TYPE E_CameraRegisters :
(
pDeviceManifestSchemaMinorVersionReg_pDeviceManifestXMLMajorVersionReg_DeviceManifestSecondaryURL_pDeviceManifestSchemaMajorVersionReg_pDeviceManifestXMLSubMinorVersionReg_pDeviceManifestXMLMinorVersionReg_DeviceManifestPrimaryURL_BootStrap_VersionMajor_BootStrap_VersionMinor := 16#00000000, // GigE Vision Minor Version
BootStrap_DeviceEndianess_BootStrap_CharacterSet_pURLRegisterAddressReg := 16#00000004, // None
BootStrap_MACAddress_High      := 16#00000008, // None
BootStrap_MACAddress_Low       := 16#0000000C, // None
BootStrap_EnabledDHCP_BootStrap_EnabledPersistentIP_BootStrap_EnabledLLA := 16#00000014, // LLA Register Enabled
BootStrap_IPAddress            := 16#00000024, // Current IP Address Register
BootStrap_SubnetMask           := 16#00000034, // Current Subnet Mask Register
BootStrap_Gateway              := 16#00000044, // Current Subnet Mask Register
DeviceVendorName               := 16#00000048, // Name of the camera vendor which is always Beckhoff Automation GmbH & Co.KG
DeviceModelName                := 16#00000068, // Displays the device model name.
DeviceVersion                  := 16#00000088, // Displays the device version which includes the firmware release and build.
DeviceSerialNumber             := 16#000000D8, // Device's serial number. This string is a unique identifier of the device.
DeviceUserID                   := 16#000000E8, // A user set ID of up to 15 characters. By default this field is set to the serial number of the camera.
GevFirstURL                    := 16#00000200, // NULL-terminated string providing the first URL to the XML device description file.
GevSecondURL                   := 16#00000400, // NULL-terminated string providing the second URL to the XML device description file.
BootStrap_NumberOfInterfaces   := 16#00000600, // Number Of Interfaces
BootStrap_PersistentIPAddress  := 16#0000064C, // Persistent IP Address Register
BootStrap_PersistentSubnetMask := 16#0000065C, // Persistent Subnet Mask Register
BootStrap_PersistentDefaultGateway := 16#0000066C, // Persistent Default Gateway Register
BootStrap_TimestampTickFrequencyHigh := 16#0000093C, // 32-MSB of the timestamp Frequency
BootStrap_TimestampTickFrequencyLow := 16#00000940, // 32-LSB of the timestamp Frequencyy
BootStrap_GevTimestampControl  := 16#00000944, // Timestamp Control Register
BootStrap_TimestampValueHigh   := 16#00000948, // 32-MSB of the timestamp Value
BootStrap_TimestampValueLow    := 16#0000094C, // 32-LSB of the timestamp Value
pGevDiscoveryAckDelayReg       := 16#00000950, // Gev Discovery Ack Delay register
BootStrap_GVSPExtendedID       := 16#00000960, // GVSP Extended ID
BootStrap_StreamChannelDestinationPort := 16#00000D00, // BootStrap Stream Channel Destination Port register
pGevSCPSDoNotFragmentReg       := 16#00000D04, // None
pGevSCPDReg                    := 16#00000D08, // Inter-Packet Delay Register
BootStrap_StreamChannelDestinationAddress := 16#00000D18, // BootStrap Stream Channel Destination Address register
BootStrap_StreamChannelSourcePort := 16#00000D1C, // BootStrap Stream Channel Source Port register
pReverseXReg                   := 16#01F81400, // None
pAcquisitionModeReg            := 16#01F83200, // None
pGevPhysicalLinkConfiguration  := 16#01F84E00, // None
pDeviceTypeReg                 := 16#01F90000, // None
pAcquisitionFrameRateEnableIsAvailableReg := 16#01F93400, // None
pEtherCATLinkActiveReg         := 16#01F93900, // None
pPayloadSizeHighReg            := 16#01F93D00, // None
pPayloadSizeLowReg             := 16#01F93D04, // None
pGevActiveLinkCountReg         := 16#01F93E00, // None
pOpticControllerPresentReg     := 16#01F94500, // None
pLightControllerPresentReg     := 16#01F95200, // None
pTestPatternCountReg           := 16#01FA0204, // None
pOpticControllerStatusReg      := 16#01FA1100, // None
pLightControllerPowerGoodReg   := 16#01FA1300, // None
pReverseYReg                   := 16#02F81400, // None
pAcquisitionStartReg           := 16#02F83200, // None
pGainBaseReg                   := 16#02F84600, // None
pDigitalAllGainReg             := 16#02F84604, // None
pDigitalRedGainReg             := 16#02F84608, // None
pDigitalGreenGainReg           := 16#02F8460C, // None
pDigitalBlueGainReg            := 16#02F84610, // None
pGevCurrentPhysicalLinkConfiguration := 16#02F84E00, // None
pTemperatureCompensationModeReg := 16#02F86C00, // None
pLightControllerEnabledReg     := 16#02F87D00, // None
pDeviceScanTypeReg             := 16#02F90000, // None
pAcquisitionFrameRateIsAvailableReg := 16#02F93400, // None
pEtherCATStateReg              := 16#02F93900, // None
pTransferBlockDurationHighReg  := 16#02F93B00, // None
pTransferBlockDurationLowReg   := 16#02F93B04, // None
pApertureReg                   := 16#02F94500, // Aperture Register
pLightConnectionStatusReg      := 16#02F95200, // None
pDeviceTemperatureImageSensorReg := 16#02FA0000, // None
pDeviceTemperatureCoreReg      := 16#02FA0004, // None
pDeviceTemperatureEthernetPhyReg := 16#02FA0008, // None
pDeviceTemperatureLiquidLensReg := 16#02FA000C, // None
TestPatternDescription         := 16#02FA0200, // None
pLightController0Channel0TriggerActiveReg := 16#02FA1300, // Trigger selected channel active register
pLightController0Channel1TriggerActiveReg := 16#02FA1304, // Trigger channel 1 active register
pLightController0Channel2TriggerActiveReg := 16#02FA1308, // Trigger channel 2 active register
pLightController0Channel3TriggerActiveReg := 16#02FA130C, // Trigger channel 3 active register
pPixelFormatReg                := 16#03F81400, // None
pAcquisitionStopReg            := 16#03F83200, // None
pMinimumObjectCameraDistanceReg := 16#03F83504, // Minimum Object Camera Distance Register
pMaximumObjectCameraDistanceReg := 16#03F83508, // Maximum Object Camera Distance Register
pObjectCameraDistanceReg       := 16#03F86C00, // Object Camera Distance Register
pPhysicalWidthReg              := 16#03F92600, // None
pGevSupportedOptionHighWordReg := 16#03F93E00, // None
pGevSupportedOptionLowWordReg  := 16#03F93E04, // None
pNumericalApertureReg          := 16#03F94500, // Numerical Aperture Register
pTestPatternReg                := 16#03FA0200, // None
pDecimationImplementedReg      := 16#04F81400, // None
pDecimationModesCapabilityReg  := 16#04F81404, // None
pDecimationHorizontalFactorsCapabilityReg := 16#04F81408, // None
pDecimationVerticalFactorsCapabilityReg := 16#04F8140C, // None
pAcquisitionAbortReg           := 16#04F83200, // None
pBlackLevelReg                 := 16#04F84600, // None
pGevPAUSEFrameReception        := 16#04F84E00, // None
pLensCalibrationModeReg        := 16#04F86C00, // Lens Calibration Mode Register
LightController0Channel0ColorDescription := 16#04F87D00, // The color of the emitted light.
LightController0Channel1ColorDescription := 16#04F87D20, // The color of the emitted light.
LightController0Channel2ColorDescription := 16#04F87D40, // The color of the emitted light.
LightController0Channel3ColorDescription := 16#04F87D60, // The color of the emitted light.
pPhysicalHeightReg             := 16#04F92600, // None
pAcquisitionStatusAcquisitionTriggerWaitReg := 16#04F93400, // None
pAcquisitionStatusAcquisitionActiveReg := 16#04F93404, // None
pGevMACAddressHighWordReg      := 16#04F93E00, // None
pFocalPowerReg                 := 16#04F94500, // Focal Power Register
pTestPatternModeReg            := 16#04FA0200, // None
pDeviceLink0ThroughputLimitModeReg := 16#05F80000, // None
pDeviceLink1ThroughputLimitModeReg := 16#05F80040, // None
pDecimationHorizontalModeReg   := 16#05F81400, // None
pAcquisitionFrameCountReg      := 16#05F83200, // None
pBlackLevelAutoReg             := 16#05F84600, // None
pGevPAUSEFrameTransmission     := 16#05F84E00, // None
pLensCalibrationStepNearReg    := 16#05F86C00, // None
pLightController0Channel0BrightnessReg := 16#05F87D00, // Light Controller0 Channel0 Brightness register
pLightController0Channel1BrightnessReg := 16#05F87D04, // Light Controller0 Channel1 Brightness register
pLightController0Channel2BrightnessReg := 16#05F87D08, // Light Controller0 Channel2 Brightness register
pLightController0Channel3BrightnessReg := 16#05F87D0C, // Light Controller0 Channel3 Brightness register
DeviceFamilyName               := 16#05F90000, // Displays the family of the camera model.
pSensorPixelWidthReg           := 16#05F92600, // None
pLineTriggerAvailableReg       := 16#05F93400, // None
pGevMACAddressLowWordReg       := 16#05F93E00, // None
pObjectSensorDistanceReg       := 16#05F94500, // Object Sensor Distance Register
pTestPatternParameter1Reg      := 16#05FA0200, // None
pDeviceLink0ThroughputLimitRatioReg := 16#06F80000, // None
pDeviceLink1ThroughputLimitRatioReg := 16#06F80040, // None
pDeviceLinkMinimumThroughputLimitRatioReg := 16#06F80044, // None
pDecimationHorizontalReg       := 16#06F81400, // None
pAcquisitionFrameRateEnableReg := 16#06F83200, // None
pLensCalibrationStepFarReg     := 16#06F86C00, // None
pLightController0Channel0BrightnessMinimumReg := 16#06F87D00, // Light Controller0 Channel0 Brightness Minimum register
pLightController0Channel1BrightnessMinimumReg := 16#06F87D04, // Light Controller0 Channel1 Brightness Minimum register
pLightController0Channel2BrightnessMinimumReg := 16#06F87D08, // Light Controller0 Channel2 Brightness Minimum register
pLightController0Channel3BrightnessMinimumReg := 16#06F87D0C, // Light Controller0 Channel3 Brightness Minimum register
DeviceManufacturerInfo         := 16#06F90000, // Manufactuer information about the device.
pSensorPixelHeightReg          := 16#06F92600, // None
pGevIPConfigurationStatusReg   := 16#06F93E00, // None
pFocalLengthReg                := 16#06F94500, // Focal Length Register
pTestPatternParameter2Reg      := 16#06FA0200, // None
pDeviceLink0ThroughputLimitReg := 16#07F80000, // None
pDeviceLink1ThroughputLimitReg := 16#07F80040, // None
pDecimationHorizontalMinimumReg := 16#07F81400, // None
pFrameRateReg                  := 16#07F83200, // None
pBalanceRatioReg               := 16#07F84600, // None
pBalanceRatioRedReg            := 16#07F84604, // None
pBalanceRatioGreenReg          := 16#07F84608, // None
pBalanceRatioBlueReg           := 16#07F8460C, // None
pLensCalibrationCoefficient1Reg := 16#07F86C00, // Lens Calibration Coefficient 1 Register
pLightController0Channel0BrightnessMaximumReg := 16#07F87D00, // Light Controller0 Channel0 Brightness Maximum register
pLightController0Channel1BrightnessMaximumReg := 16#07F87D04, // Light Controller0 Channel1 Brightness Maximum register
pLightController0Channel2BrightnessMaximumReg := 16#07F87D08, // Light Controller0 Channel2 Brightness Maximum register
pLightController0Channel3BrightnessMaximumReg := 16#07F87D0C, // Light Controller0 Channel3 Brightness Maximum register
SensorName                     := 16#07F92600, // Displays the model of the sensor.
pMagnificationReg              := 16#07F94500, // Magnification Register
pTestPatternHorizontalPositionReg := 16#07FA0200, // None
pDeviceLink0HeartbeatModeReg   := 16#08F80000, // None
pDeviceLink1HeartbeatModeReg   := 16#08F80040, // None
pDecimationHorizontalMaximumReg := 16#08F81400, // None
pFrameRateRegMaxReg            := 16#08F83200, // None
pGammaReg                      := 16#08F84600, // None
pLensCalibrationCoefficient2Reg := 16#08F86C00, // Lens Calibration Coefficient 2 Register
pLightController0Channel0TriggerModeReg := 16#08F87D00, // Light Controller0 Channel0 Trigger Mode register
pLightController0Channel1TriggerModeReg := 16#08F87D04, // Light Controller0 Channel1 Trigger Mode register
pLightController0Channel2TriggerModeReg := 16#08F87D08, // Light Controller0 Channel2 Trigger Mode register
pLightController0Channel3TriggerModeReg := 16#08F87D0C, // Light Controller0 Channel3 Trigger Mode register
DeviceFirmwareVersion          := 16#08F90000, // Displays the currently loaded firmware version manufacturer's code.
pSensorShutterModeReg          := 16#08F92600, // None
pFieldOfViewHorizontalReg      := 16#08F94500, // Field Of View Horizontal Register
pTestPatternVerticalPositionReg := 16#08FA0200, // None
pDeviceLink0HeartbeatTimeoutReg := 16#09F80000, // None
pDeviceLink1HeartbeatTimeoutReg := 16#09F80040, // None
pDecimationVerticalModeReg     := 16#09F81400, // None
pFrameRateRegMinReg            := 16#09F83200, // None
pLensCalibrationCoefficient3Reg := 16#09F86C00, // Lens Calibration Coefficient 3 Register
pLightController0Channel0TriggerDurationReg := 16#09F87D00, // Light Controller0 Channel0 Trigger Duration register
pLightController0Channel1TriggerDurationReg := 16#09F87D04, // Light Controller0 Channel1 Trigger Duration register
pLightController0Channel2TriggerDurationReg := 16#09F87D08, // Light Controller0 Channel2 Trigger Duration register
pLightController0Channel3TriggerDurationReg := 16#09F87D0C, // Light Controller0 Channel3 Trigger Duration register
pRegionsPresentReg             := 16#09F92600, // Maximum regions of interest present.
pFieldOfViewVerticalReg        := 16#09F94500, // Field Of View Vertical Register
pTestPatternHorizontalStepSizeReg := 16#09FA0200, // None
pDecimationVerticalReg         := 16#0AF81400, // None
pLensCalibrationCoefficient4Reg := 16#0AF86C00, // Lens Calibration Coefficient 4 Register
pLightController0Channel0TriggerDelayReg := 16#0AF87D00, // Light Controller0 Channel0 Trigger Delay register
pLightController0Channel1TriggerDelayReg := 16#0AF87D04, // Light Controller0 Channel1 Trigger Delay register
pLightController0Channel2TriggerDelayReg := 16#0AF87D08, // Light Controller0 Channel2 Trigger Delay register
pLightController0Channel3TriggerDelayReg := 16#0AF87D0C, // Light Controller0 Channel3 Trigger Delay register
pDeviceSFNCVersionMajorReg     := 16#0AF90000, // None
pPixelSizeReg                  := 16#0AF92600, // None
pFieldOfViewDiagonalReg        := 16#0AF94500, // Field Of View Diagonal Register
pTestPatternVerticalStepSizeReg := 16#0AFA0200, // None
pDecimationVerticalMinimumReg  := 16#0BF81400, // None
pLensCalibrationCoefficient5Reg := 16#0BF86C00, // Lens Calibration Coefficient 5 Register
pDeviceSFNCVersionMinorReg     := 16#0BF90000, // None
pPixelColorFilterReg           := 16#0BF92600, // None
pDepthOfFieldReg               := 16#0BF94500, // Depth Of Field Register
pTestPatternHorizontalNumReg   := 16#0BFA0200, // None
pDeviceResetReg                := 16#0CF80000, // None
pDecimationVerticalMaximumReg  := 16#0CF81400, // None
pTriggerModeAcquisitionStartReg := 16#0CF83200, // None
pTriggerModeFrameStartReg      := 16#0CF8320C, // None
pLensTemperatureCalibrationCoefficient1Reg := 16#0CF86C00, // Lens Temperature Calibration Coefficient 1 Register
pDeviceSFNCVersionSubMinorReg  := 16#0CF90000, // None
pPixelFilterArrayReg           := 16#0CF92600, // None
pDepthOfFieldNearReg           := 16#0CF94500, // Depth Of Field Near Register
pTestPatternVerticalNumReg     := 16#0CFA0200, // None
pDeviceIndicatorModeReg        := 16#0DF80000, // None
pSoftwareTriggerAcquisitionStartReg := 16#0DF83200, // None
pSoftwareTriggerFrameStartReg  := 16#0DF8320C, // None
pLensTemperatureCalibrationCoefficient2Reg := 16#0DF86C00, // Lens Temperature Calibration Coefficient 2 Register
pDeviceTLTypeReg               := 16#0DF90000, // None
pSensorColorReg                := 16#0DF92600, // True, if a color sensor has been detected.
pDepthOfFieldFarReg            := 16#0DF94500, // Depth Of Field Far Register
pTestPatternColorWidthReg      := 16#0DFA0200, // None
pDeviceRegisterCheckReg        := 16#0EF80000, // None
pRegion0ModeReg                := 16#0EF81400, // Region Mode 0 register.
pRegion1ModeReg                := 16#0EF81404, // Region Mode 1 register.
pRegion2ModeReg                := 16#0EF81408, // Region Mode 2 register.
pRegion3ModeReg                := 16#0EF8140C, // Region Mode 3 register.
pRegion4ModeReg                := 16#0EF81410, // Region Mode 4 register.
pRegion5ModeReg                := 16#0EF81414, // Region Mode 5 register.
pRegion6ModeReg                := 16#0EF81418, // Region Mode 6 register.
pRegion7ModeReg                := 16#0EF8141C, // Region Mode 7 register.
pTriggerSourceSoftwareReg      := 16#0EF83200, // None
pTriggerSourceFrameStartReg    := 16#0EF8320C, // None
pLensTemperatureCalibrationCoefficient3Reg := 16#0EF86C00, // Lens Temperature Calibration Coefficient 3 Register
pDeviceTLVersionMajorReg       := 16#0EF90000, // None
pSensorPolarizationReg         := 16#0EF92600, // True, if a polarization sensor has been detected.
pTestPatternBackGroundReg      := 16#0EFA0200, // None
pDeviceRegisterValidReg        := 16#0FF80000, // None
pRegion0WidthReg               := 16#0FF81400, // None
pRegion1WidthReg               := 16#0FF81404, // None
pRegion2WidthReg               := 16#0FF81408, // None
pRegion3WidthReg               := 16#0FF8140C, // None
pRegion4WidthReg               := 16#0FF81410, // None
pRegion5WidthReg               := 16#0FF81414, // None
pRegion6WidthReg               := 16#0FF81418, // None
pRegion7WidthReg               := 16#0FF8141C, // None
pTriggerActivationAcquisitionStartReg := 16#0FF83200, // None
pTriggerActivationFrameStartReg := 16#0FF8320C, // None
pForceIPAddressReg             := 16#0FF84E00, // Force IP Address Register
pLoadLensCalibrationSettingsReg := 16#0FF86C00, // None
pDeviceTLVersionMinorReg       := 16#0FF90000, // None
pTestPatternGradientStepReg    := 16#0FFA0200, // None
pTestPatternParameterMaskReg   := 16#0FFA0208, // None
pRegion0MinWidthReg            := 16#10F81400, // None
pRegion1MinWidthReg            := 16#10F81404, // None
pRegion2MinWidthReg            := 16#10F81408, // None
pRegion3MinWidthReg            := 16#10F8140C, // None
pRegion4MinWidthReg            := 16#10F81410, // None
pRegion5MinWidthReg            := 16#10F81414, // None
pRegion6MinWidthReg            := 16#10F81418, // None
pRegion7MinWidthReg            := 16#10F8141C, // None
pTriggerDelayAcquisitionStartReg := 16#10F83200, // None
pTriggerDelayFrameStartReg     := 16#10F8320C, // None
pForceSubnetMaskReg            := 16#10F84E00, // Force Subnet Mask Register
pSaveLensCalibrationSettingsReg := 16#10F86C00, // None
pDeviceTLVersionSubMinorReg    := 16#10F90000, // None
pDeviceClockBaseReg            := 16#11F80000, // None
pRegion0MaxWidthReg            := 16#11F81400, // None
pRegion1MaxWidthReg            := 16#11F81404, // None
pRegion2MaxWidthReg            := 16#11F81408, // None
pRegion3MaxWidthReg            := 16#11F8140C, // None
pRegion4MaxWidthReg            := 16#11F81410, // None
pRegion5MaxWidthReg            := 16#11F81414, // None
pRegion6MaxWidthReg            := 16#11F81418, // None
pRegion7MaxWidthReg            := 16#11F8141C, // None
pExposureModeReg               := 16#11F83200, // None
pForceDefaultGatewayReg        := 16#11F84E00, // Force Default Gateway Register
pRestoreLensCalibrationFactorySettingsReg := 16#11F86C00, // None
pMaxThroughputReg              := 16#11F90000, // None
pTimestampActiveSourceReg      := 16#12F80000, // None
pRegion0IncWidthReg            := 16#12F81400, // None
pRegion1IncWidthReg            := 16#12F81404, // None
pRegion2IncWidthReg            := 16#12F81408, // None
pRegion3IncWidthReg            := 16#12F8140C, // None
pRegion4IncWidthReg            := 16#12F81410, // None
pRegion5IncWidthReg            := 16#12F81414, // None
pRegion6IncWidthReg            := 16#12F81418, // None
pRegion7IncWidthReg            := 16#12F8141C, // None
pExposureTimeReg               := 16#12F83200, // None
pForceIPActivateReg            := 16#12F84E00, // None
pDeviceStateReg                := 16#13F80000, // None
pRegion0HeightReg              := 16#13F81400, // None
pRegion1HeightReg              := 16#13F81404, // None
pRegion2HeightReg              := 16#13F81408, // None
pRegion3HeightReg              := 16#13F8140C, // None
pRegion4HeightReg              := 16#13F81410, // None
pRegion5HeightReg              := 16#13F81414, // None
pRegion6HeightReg              := 16#13F81418, // None
pRegion7HeightReg              := 16#13F8141C, // None
pExposureTimeMaxReg            := 16#13F83200, // None
pDeviceConnection0SpeedReg     := 16#13F90000, // None
pDeviceConnection1SpeedReg     := 16#13F90004, // None
pDeviceDefaultStateReg         := 16#14F80000, // None
pRegion0MinHeightReg           := 16#14F81400, // None
pRegion1MinHeightReg           := 16#14F81404, // None
pRegion2MinHeightReg           := 16#14F81408, // None
pRegion3MinHeightReg           := 16#14F8140C, // None
pRegion4MinHeightReg           := 16#14F81410, // None
pRegion5MinHeightReg           := 16#14F81414, // None
pRegion6MinHeightReg           := 16#14F81418, // None
pRegion7MinHeightReg           := 16#14F8141C, // None
pExposureTimeMinReg            := 16#14F83200, // None
pDeviceConnection0StatusReg    := 16#14F90000, // None
pDeviceConnection1StatusReg    := 16#14F90004, // None
pRegion0MaxHeightReg           := 16#15F81400, // None
pRegion1MaxHeightReg           := 16#15F81404, // None
pRegion2MaxHeightReg           := 16#15F81408, // None
pRegion3MaxHeightReg           := 16#15F8140C, // None
pRegion4MaxHeightReg           := 16#15F81410, // None
pRegion5MaxHeightReg           := 16#15F81414, // None
pRegion6MaxHeightReg           := 16#15F81418, // None
pRegion7MaxHeightReg           := 16#15F8141C, // None
pRegion0IncHeightReg           := 16#16F81400, // None
pRegion1IncHeightReg           := 16#16F81404, // None
pRegion2IncHeightReg           := 16#16F81408, // None
pRegion3IncHeightReg           := 16#16F8140C, // None
pRegion4IncHeightReg           := 16#16F81410, // None
pRegion5IncHeightReg           := 16#16F81414, // None
pRegion6IncHeightReg           := 16#16F81418, // None
pRegion7IncHeightReg           := 16#16F8141C, // None
pGevSCPInterfaceIndexReg       := 16#16F84E00, // Gev SCP Interface Index Register
pDeviceLink0SpeedReg           := 16#16F90000, // None
pDeviceLink1SpeedReg           := 16#16F90040, // None
pRegion0OffsetXReg             := 16#17F81400, // None
pRegion1OffsetXReg             := 16#17F81404, // None
pRegion2OffsetXReg             := 16#17F81408, // None
pRegion3OffsetXReg             := 16#17F8140C, // None
pRegion4OffsetXReg             := 16#17F81410, // None
pRegion5OffsetXReg             := 16#17F81414, // None
pRegion6OffsetXReg             := 16#17F81418, // None
pRegion7OffsetXReg             := 16#17F8141C, // None
pGevSCPSPacketSizeReg          := 16#17F84E00, // None
pGevSCPSPacketSizeMinReg       := 16#17F84E04, // Minimum packet size register
pGevSCPSPacketSizeMaxReg       := 16#17F84E08, // Maximum packet size register
pGevSCPSPacketSizeIncReg       := 16#17F84E0C, // Increment of packet size register
pDeviceLink0ConnectionCountReg := 16#17F90000, // None
pDeviceLink1ConnectionCountReg := 16#17F90040, // None
pRegion0MinOffsetXReg          := 16#18F81400, // None
pRegion1MinOffsetXReg          := 16#18F81404, // None
pRegion2MinOffsetXReg          := 16#18F81408, // None
pRegion3MinOffsetXReg          := 16#18F8140C, // None
pRegion4MinOffsetXReg          := 16#18F81410, // None
pRegion5MinOffsetXReg          := 16#18F81414, // None
pRegion6MinOffsetXReg          := 16#18F81418, // None
pRegion7MinOffsetXReg          := 16#18F8141C, // None
pDeviceStreamChannelCount      := 16#18F90000, // None
pRegion0MaxOffsetXReg          := 16#19F81400, // None
pRegion1MaxOffsetXReg          := 16#19F81404, // None
pRegion2MaxOffsetXReg          := 16#19F81408, // None
pRegion3MaxOffsetXReg          := 16#19F8140C, // None
pRegion4MaxOffsetXReg          := 16#19F81410, // None
pRegion5MaxOffsetXReg          := 16#19F81414, // None
pRegion6MaxOffsetXReg          := 16#19F81418, // None
pRegion7MaxOffsetXReg          := 16#19F8141C, // None
pRegion0IncOffsetXReg          := 16#1AF81400, // None
pRegion1IncOffsetXReg          := 16#1AF81404, // None
pRegion2IncOffsetXReg          := 16#1AF81408, // None
pRegion3IncOffsetXReg          := 16#1AF8140C, // None
pRegion4IncOffsetXReg          := 16#1AF81410, // None
pRegion5IncOffsetXReg          := 16#1AF81414, // None
pRegion6IncOffsetXReg          := 16#1AF81418, // None
pRegion7IncOffsetXReg          := 16#1AF8141C, // None
pDeviceStreamChannel1StateReg  := 16#1AF90000, // None
pDeviceStreamChannel2StateReg  := 16#1AF90040, // None
pRegion0OffsetYReg             := 16#1BF81400, // None
pRegion1OffsetYReg             := 16#1BF81404, // None
pRegion2OffsetYReg             := 16#1BF81408, // None
pRegion3OffsetYReg             := 16#1BF8140C, // None
pRegion4OffsetYReg             := 16#1BF81410, // None
pRegion5OffsetYReg             := 16#1BF81414, // None
pRegion6OffsetYReg             := 16#1BF81418, // None
pRegion7OffsetYReg             := 16#1BF8141C, // None
pDeviceStreamChannel1TypeReg   := 16#1BF90000, // None
pDeviceStreamChannel2TypeReg   := 16#1BF90040, // None
pRegion0MinOffsetYReg          := 16#1CF81400, // None
pRegion1MinOffsetYReg          := 16#1CF81404, // None
pRegion2MinOffsetYReg          := 16#1CF81408, // None
pRegion3MinOffsetYReg          := 16#1CF8140C, // None
pRegion4MinOffsetYReg          := 16#1CF81410, // None
pRegion5MinOffsetYReg          := 16#1CF81414, // None
pRegion6MinOffsetYReg          := 16#1CF81418, // None
pRegion7MinOffsetYReg          := 16#1CF8141C, // None
pGevSCPDMinReg                 := 16#1CF84E00, // Minimum Inter-Packet Delay register
pGevSCPDMaxReg                 := 16#1CF84E04, // Maximum Inter-Packet Delay register
pGevSCPDIncReg                 := 16#1CF84E08, // Increment Inter-Packet Delay register
pDeviceStreamChannel1LinkReg   := 16#1CF90000, // None
pDeviceStreamChannel2LinkReg   := 16#1CF90040, // None
pRegion0MaxOffsetYReg          := 16#1DF81400, // None
pRegion1MaxOffsetYReg          := 16#1DF81404, // None
pRegion2MaxOffsetYReg          := 16#1DF81408, // None
pRegion3MaxOffsetYReg          := 16#1DF8140C, // None
pRegion4MaxOffsetYReg          := 16#1DF81410, // None
pRegion5MaxOffsetYReg          := 16#1DF81414, // None
pRegion6MaxOffsetYReg          := 16#1DF81418, // None
pRegion7MaxOffsetYReg          := 16#1DF8141C, // None
pDeviceStreamChannel1EndiannessReg := 16#1DF90000, // None
pDeviceStreamChannel2EndiannessReg := 16#1DF90040, // None
pRegion0IncOffsetYReg          := 16#1EF81400, // None
pRegion1IncOffsetYReg          := 16#1EF81404, // None
pRegion2IncOffsetYReg          := 16#1EF81408, // None
pRegion3IncOffsetYReg          := 16#1EF8140C, // None
pRegion4IncOffsetYReg          := 16#1EF81410, // None
pRegion5IncOffsetYReg          := 16#1EF81414, // None
pRegion6IncOffsetYReg          := 16#1EF81418, // None
pRegion7IncOffsetYReg          := 16#1EF8141C, // None
pDeviceStreamChannel1PacketSizeReg := 16#1EF90000, // None
pDeviceStreamChannel2PacketSizeReg := 16#1EF90040, // None
pDeviceEventChannelCountReg    := 16#20F90000, // None
pDeviceCharacterSetReg         := 16#21F90000, // None
pDeviceRegistersEndiannessReg  := 16#22F90000, // None
pTimestampHighReg              := 16#23F90000, // None
pTimestampRegLow               := 16#23F90004, // None
pExtendedInternalTimestampControlRegister := 16#25F90000, // None
pTimestampLatchRegHighReg      := 16#26F90000, // None
pTimestampLatchLowReg          := 16#26F90004, // None
UserSetDescription             := 16#30001120, // Description of the selected User Set content.
UserSetDescription1            := 16#30001140, // Description of the selected User Set content.
UserSetDescription2            := 16#30001160, // Description of the selected User Set content.
UserSetDescription3            := 16#30001180, // Description of the selected User Set content.
UserSetDescription4            := 16#300011A0, // Description of the selected User Set content.
pUserSet0LoadReg               := 16#30001200, // None
pUserSet1LoadReg               := 16#30001204, // None
pUserSet2LoadReg               := 16#30001208, // None
pUserSet3LoadReg               := 16#3000120C, // None
pUserSet4LoadReg               := 16#30001210, // None
pUserSet0SaveReg               := 16#30001300, // None
pUserSet1SaveReg               := 16#30001304, // None
pUserSet2SaveReg               := 16#30001308, // None
pUserSet3SaveReg               := 16#3000130C, // None
pUserSet4SaveReg               := 16#30001310, // None
pUserSetDefaultReg             := 16#30001500, // None
pUserSetFeatureEnableReg       := 16#30001510, // None
pUserSetMaxFeatures            := 16#30001514, // None
pLineModeReg                   := 16#30020040, // None
pLineInverterReg               := 16#30030040, // None
pLineStatus                    := 16#30040040, // None
pHorizontalBinningReg          := 16#31001030, // None
pVerticalBinningReg            := 16#31001034, // None
pLUTEnabledReg                 := 16#35000000, // None
pCounter0EventSourceReg        := 16#37000100, // Counter0 Event Source Reg
pCounter1EventSourceReg        := 16#37000104, // Counter1 Event Source Reg
pCounter2EventSourceReg        := 16#37000108, // Counter2 Event Source Reg
pCounter3EventSourceReg        := 16#3700010C, // Counter3 Event Source Reg
pCounter4EventSourceReg        := 16#37000110, // Counter4 Event Source Reg
pCounter5EventSourceReg        := 16#37000114, // Counter5 Event Source Reg
pCounter0ResetReg              := 16#37000200, // Counter0 Reset Reg
pCounter1ResetReg              := 16#37000204, // Counter1 Reset Reg
pCounter2ResetReg              := 16#37000208, // Counter2 Reset Reg
pCounter3ResetReg              := 16#3700020C, // Counter3 Reset Reg
pCounter4ResetReg              := 16#37000210, // Counter4 Reset Reg
pCounter5ResetReg              := 16#37000214, // Counter5 Reset Reg
pCounter0ValueReg              := 16#37000300, // Counter0 Value Reg
pCounter1ValueReg              := 16#37000304, // Counter1 Value Reg
pCounter2ValueReg              := 16#37000308, // Counter2 Value Reg
pCounter3ValueReg              := 16#3700030C, // Counter3 Value Reg
pCounter4ValueReg              := 16#37000310, // Counter4 Value Reg
pCounter5ValueReg              := 16#37000314 // Counter5 Value Reg
) UDINT;
END_TYPE

(* stored: Version 1.1.0.1, ProductVersion 3.1.4024.7
   DUT E_CameraRegisters: Id {e8aa0ed4-75b7-4c9a-ab87-f5047f3dbf61} *)
